# B&R Automation Studio project CentralEne
Automation Studio 4.4.4.112; technology packages: Acp10Arnc0 3.18.2, mapp 1.64.1, mappControl 5.1.0, mappView 5.1.1

## Configuration Central

CPU X20CP1301, AutomationRuntime F4.44, Build 4.1.2, Vc V4.44.0

### Task classes (Cpu.sw)
```
Cyclic#6:
  acionaSina <- Programa.acionaSinais.prg
  preparaDet <- Programa.preparaDetectores.prg
Cyclic#7:
  transmiteD <- Programa.transmiteDetectores.prg
DataObjects: Acp10sys
VcDataObjects: Visu <- Programa.Visu.dob
Binaries: TCData, vccalarm, vcnet, vcrt, vcpkat, vcctext, vctcal, vcfile, vcgclass, vcctrend, Visu03, vcpdsw, arial, vccbmp, vcmgr, vcchspot, vcdsloc, vcfntttf, Visu02, vccovl, vcshared, arialbd, vcalarm, vccdt, vccline, vccbtn, vcpdvnc, vcbclass, vcpfx20, vcdsint, vccnum, Visu01, mvLoader, udbdef, ashwac, Role, ashwd, arconfig, sysconf, iomap, User, asfw, Acp10map, acp10cfg, vcpfar00
Libraries: AsHttp, runtime, standard, LoopConR, sys_lib, brsystem, Acp10par, NcGlobal, Acp10man, asieccon, astime, vcresman, fileio, ashw, dataobj, powerlnk
```

### Hardware
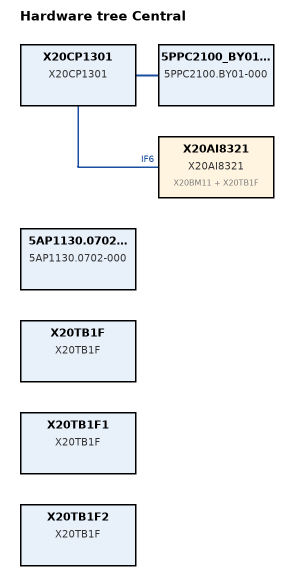
```
5AP1130.0702-000 : 5AP1130.0702-000 v1.3.0.0
  Terminal = true
  Mode = Manual
  InternetAddress = 172.21.12.120
  DefaultGateway = 172.21.12.2
  SubnetMask = 255.255.255.0
5PPC2100_BY01_000 : 5PPC2100.BY01-000 v1.2.9.0  [IF3 -> X20CP1301.IF2 [Cable Type=PowerlinkCable, Length=10, Version=1.0.0.2]; SY -> 5AP1130.0702-000.SY1]
  Connector IF3
  Terminal = true
X20AI8321 : X20AI8321 v1.3.0.0  [SS1 -> X20TB1F3.SS; SL -> X20BM11.SL1]
  LowerLimit = 0
  ChannelType01 = 4 to 20mA
  ChannelType02 = 4 to 20mA
  ChannelType03 = 4 to 20mA
  ChannelType04 = 4 to 20mA
  ChannelType05 = 4 to 20mA
X20BM11 : X20BM11 v1.0.0.1  [X2X1 -> X20CP1301.IF6]
X20CP1301 : X20CP1301 v1.6.1.0  [X1 -> X1.SL; X2 -> X2.SL; X3 -> X3.SL]
  Module X1 (Type=X1, Virtual=true, Version=1.6.1.0)
    Connection (Connector=SS1, TargetModule=X20TB1F, TargetConnector=SS)
    Connection (Connector=SL, TargetModule=X20CP1301, TargetConnector=X1)
  Module X2 (Type=X2, Virtual=true, Version=1.6.1.0)
    Connection (Connector=SS1, TargetModule=X20TB1F1, TargetConnector=SS)
    Connection (Connector=SL, TargetModule=X20CP1301, TargetConnector=X2)
  Module X3 (Type=X3, Virtual=true, Version=1.6.1.0)
    Connection (Connector=SS1, TargetModule=X20TB1F2, TargetConnector=SS)
    Connection (Connector=SL, TargetModule=X20CP1301, TargetConnector=X3)
  Connector IF2:
    ActivateDevice = 1
    HostName = loga
    Mode = Manual
    InternetAddress = 172.21.12.119
    SubnetMask = 255.255.255.0
    Vnc1
    VncVcObjectName1 = Visu
    VncKeyMappingFile1 = VC\PS2-Keyboard.dis
    VncAuthentication1 = 1
    VncPasswordViewOnly1 = v
    VncPasswordViewControl1 = c
  ConfigurationID = CentralEne_Central
  EthernetDefaultGateway = 172.21.12.2
  ActivateDns = 1
  DnsServer1 = 172.21.4.143
X20TB1F : X20TB1F v1.0.0.0
X20TB1F1 : X20TB1F v1.0.0.0
X20TB1F2 : X20TB1F v1.0.0.0
X20TB1F3 : X20TB1F v1.0.0.0
```

### IoMap.iom - X20CP1301/IoMap.iom
```iecst
VAR_CONFIG
	::preparaDet:aiDG[1] AT %IW."X20AI8321".AnalogInput01;
	::preparaDet:aiDG[2] AT %IW."X20AI8321".AnalogInput02;
	::preparaDet:aiDG[3] AT %IW."X20AI8321".AnalogInput03;
	::preparaDet:aiDG[5] AT %IW."X20AI8321".AnalogInput04;
	::preparaDet:aiDG[4] AT %IW."X20AI8321".AnalogInput05;
	::Estrutura.do01SinVd AT %QX."X3".DigitalOutput01;
	::Estrutura.do02SinAm AT %QX."X3".DigitalOutput02;
	::Estrutura.do03SinVm AT %QX."X3".DigitalOutput03;
	::Estrutura.do04SinVd AT %QX."X3".DigitalOutput04;
	::Estrutura.do05SinAm AT %QX."X3".DigitalOutput05;
	::Estrutura.do06SinVm AT %QX."X3".DigitalOutput06;
	::Estrutura.do07Buzer AT %QX."X3".DigitalOutput07;
	::Estrutura.do08Modem AT %QX."X3".DigitalOutput08;
END_VAR
```

### Acp10cfg.ncc - X20CP1301/Motion/Acp10cfg.ncc
```
NcConfiguration (Version=3.18.2, NcSwId=Acp10)
  ACP10CF1_typ:
    cnt_nettrc_rec_drive = 150
    bufsize_trace_upload = 1200
    tc_nc_man_task = Cyclic #1
    glob_pv_as_ncobject = Yes
    ncsys_dl_broadcast = Yes
    ncsys_dl_acp_reset = Yes
    safemc_log_err_to_ax = Yes
    network_init:
      ncsw_init_execute = Yes
      automatic_execute = No
      node_nr_warning = Yes
      net_err_before_ncact = Yes
    nettrc:
      enter_parsecrec = Yes
      enter_ncaction = Yes
      save_ring_startidx = No
    cam_prof_download:
      cam_dat_dl_parallel = No
      tc_cam_dl_parallel = Task class for NC Manager task
```

## Logical view

Binary libraries used (declarations not repeated): operator, runtime, astime, AsIecCon, AsHttp, standard, LoopConR 4.01.0, sys_lib, brsystem, Acp10par 3.18.2, Acp10man 3.18.2, NcGlobal 3.18.2

### Global.typ - Global data types
```iecst
TYPE
	TipoTransmiter : 	STRUCT
		idTxSoftware : STRING[80];
		txValueDet : REAL;
	END_STRUCT;
	TipoEstruturaDG_type : 	STRUCT
		Estatos : REAL;
		TX : STRING[80];
		visDet : USINT;
		ID : STRING[80] := '1';
		Alarme2 : BOOL;
		Alarme1 : BOOL;
		Area : USINT;
	END_STRUCT;
	TipoEstrutura : 	STRUCT
		DG : {REDUND_UNREPLICABLE} ARRAY[0..MAX_IDX_DETECTORES]OF TipoEstruturaDG_type;
		visDet01 : USINT;
		visDet02 : USINT;
		visDet03 : USINT;
		visDet04 : USINT;
		visDet05 : USINT;
		visSinVd : BOOL;
		visSinAm : BOOL;
		visSinVm : BOOL;
		do01SinVd : BOOL;
		do02SinAm : BOOL;
		do03SinVm : BOOL;
		do04SinVd : BOOL;
		do05SinAm : BOOL;
		do06SinVm : BOOL;
		do08Modem : BOOL;
		do07Buzer : BOOL;
		visNameDG1 : STRING[80];
		visNameDG2 : STRING[80];
		visNameDG3 : STRING[80];
		visNameDG4 : STRING[80];
		visNameDG5 : STRING[80];
		visModemReset : BOOL;
	END_STRUCT;
END_TYPE
```

### Global.var - Global variables
```iecst
VAR
	Transmissao : TipoTransmiter;
	Estrutura : TipoEstrutura;
END_VAR
(*CONTANTES*)
VAR CONSTANT
	MAX_IDX_DETECTORES : USINT := 5;
END_VAR
```


### Program Logical/Programa/preparaDetectores (IEC)

#### Variables.var
```iecst
VAR
	aiDG : ARRAY[0..MAX_IDX_DETECTORES] OF INT;
	LCRScal_DG : ARRAY[0..MAX_IDX_DETECTORES] OF LCRScal;
	uIdx : USINT; (*Contador auxiliar*)
END_VAR
```

#### Main.st
```iecst
PROGRAM _INIT
	(* Prepara o range dos detectores *)

	//Configura detector 1
	Estrutura.DG[1].Area 	:= 2;
	Estrutura.DG[2].Area 	:= 2;
	Estrutura.DG[3].Area 	:= 2;
	Estrutura.DG[4].Area 	:= 1;
	Estrutura.DG[5].Area 	:= 2;

	Estrutura.DG[1].ID		:= '73';
	Estrutura.DG[2].ID		:= '74';
	Estrutura.DG[3].ID		:= '75';
	Estrutura.DG[4].ID		:= '72';
	Estrutura.DG[5].ID		:= '76';

	LCRScal_DG[1].x1 := 0.0;	 //x1 e x2 não pode ser alterado, y1 e y2 é o range do detector
	LCRScal_DG[1].y1 := 0.0;
	LCRScal_DG[1].x2 := 32767.0;
	LCRScal_DG[1].y2 := 50.0;

	LCRScal_DG[2].x1 := 0.0;	 //x1 e x2 não pode ser alterado, y1 e y2 é o range do detector
	LCRScal_DG[2].y1 := 0.0;
	LCRScal_DG[2].x2 := 32767.0;
	LCRScal_DG[2].y2 := 100.0;

	LCRScal_DG[3].x1 := 0.0;	 //x1 e x2 não pode ser alterado, y1 e y2 é o range do detector
	LCRScal_DG[3].y1 := 0.0;
	LCRScal_DG[3].x2 := 32767.0;
	LCRScal_DG[3].y2 := 1000.0;

	LCRScal_DG[4].x1 := 0.0;	 //x1 e x2 não pode ser alterado, y1 e y2 é o range do detector
	LCRScal_DG[4].y1 := 0.0;
	LCRScal_DG[4].x2 := 32767.0;
	LCRScal_DG[4].y2 := 1000.0;

	LCRScal_DG[5].x1 := 0.0;	 //x1 e x2 não pode ser alterado, y1 e y2 é o range do detector
	LCRScal_DG[5].y1 := 0.0;
	LCRScal_DG[5].x2 := 32767.0;
	LCRScal_DG[5].y2 := 100.0;

END_PROGRAM

PROGRAM _CYCLIC

	FOR uIdx := 0 TO MAX_IDX_DETECTORES BY 1 DO

		(* Converte em numero real os valores da entrada analogica *)
		LCRScal_DG[uIdx].x := INT_TO_REAL(aiDG[uIdx]);

		(* Chama o bloco de função e declara nas variaveis os resultados *)
		LCRScal_DG[uIdx]();
		Estrutura.DG[uIdx].Estatos 	:= LCRScal_DG[uIdx].y;
		Estrutura.DG[uIdx].TX		:= REAL_TO_STRING (Estrutura.DG[uIdx].Estatos * 100000);

	END_FOR;

END_PROGRAM
```

### Program Logical/Programa/transmiteDetectores (IEC)

#### Types.typ
```iecst
TYPE
	MaqEstados_enum :
		(
		HTTP_STEP_DESABILITADO := 0,
		HTTP_STEP_CONCATENA,
		HTTP_STEP_ENVIA,
		HTTP_STEP_DELAY,
		HTTP_STEP_PROXIMO_DG,
		HTTP_STEP_CONCLUIDO,
		HTTP_STEP_ABORTA,
		HTTP_STEP_ERRO
		);
END_TYPE
```

#### Variables.var
```iecst
VAR
	Dosend : BOOL := TRUE;
	Doenable : BOOL := TRUE; (*Enables FUB Instance*)
END_VAR
VAR CONSTANT
	Host : STRING[80] := '201.6.243.3';
	HostPort : UINT := 8090;
END_VAR
VAR
	Responsedata : STRING[80];
	uri : STRING[80];
	input : BOOL;
	output : BOOL;
	elapsedTime : TIME;
END_VAR
(*Insert your comment here.*)
VAR
	eStep : MaqEstados_enum;
	iDG : USINT; (*Index atual do DG a ser enviado*)
	sAuxiliar : STRING[80];
	httpClient_0 : httpClient;
	bEnviar : BOOL; (*Comando para iniciar envio*)
	TON_0 : TON;
	Resposta : STRING[80];
END_VAR
```

#### Main.st
```iecst
PROGRAM _INIT

	uri     := '/api/historic/SaveByPositionUid2';

	httpClient_0.pHost 				:= ADR (Host);
	httpClient_0.hostPort			:= HostPort;
	httpClient_0.method 			:= httpMETHOD_GET;
	httpClient_0.option 			:= httpOPTION_HTTP_11;
	httpClient_0.pResponseData 		:= ADR (Responsedata);
	httpClient_0.responseDataSize	:= SIZEOF (Responsedata);
	httpClient_0.pUri    			:= ADR (sAuxiliar);

	TON_0.PT := T#15s;

END_PROGRAM

PROGRAM _CYCLIC

	CASE eStep OF

		HTTP_STEP_DESABILITADO:

			bEnviar := TRUE;

			IF(bEnviar)THEN

				//Reseta comando
				bEnviar := FALSE;
				iDG := 1;

				eStep := HTTP_STEP_CONCATENA;

			END_IF

		HTTP_STEP_CONCATENA:

			sAuxiliar				:= CONCAT(uri, CONCAT('/', CONCAT(Estrutura.DG[iDG].ID, CONCAT('/', Estrutura.DG[iDG].TX))));
			httpClient_0.enable		:= TRUE;
			httpClient_0.send		:= TRUE;

			eStep := HTTP_STEP_ENVIA;

		HTTP_STEP_ENVIA:

			//Checa status do bloco
			IF(httpClient_0.status <> 65535)THEN

				IF(httpClient_0.status = 0)THEN

					//Reseta comandos
					httpClient_0.send	:= FALSE;
					TON_0.IN := TRUE;

					eStep := HTTP_STEP_DELAY;
				ELSE
					eStep := HTTP_STEP_ERRO;
				END_IF
			ELSE
				eStep := HTTP_STEP_ERRO;
			END_IF

		HTTP_STEP_DELAY:

			IF(TON_0.Q)THEN

				TON_0.IN := FALSE;
				eStep := HTTP_STEP_PROXIMO_DG;

			END_IF

		HTTP_STEP_PROXIMO_DG:

			iDG := iDG + 1;

			IF(iDG > MAX_IDX_DETECTORES)THEN
				eStep := HTTP_STEP_CONCLUIDO;
			ELSE
				eStep := HTTP_STEP_CONCATENA;
			END_IF

		HTTP_STEP_CONCLUIDO:

			httpClient_0.enable := FALSE;
			httpClient_0.send	:= FALSE;
			TON_0.IN := FALSE;

			eStep := HTTP_STEP_DESABILITADO;

		HTTP_STEP_ABORTA:

			//Reseta blocos
			httpClient_0.enable := FALSE;
			httpClient_0.send	:= FALSE;
			TON_0.IN := FALSE;
			eStep := HTTP_STEP_DESABILITADO;

		HTTP_STEP_ERRO:

			//Reseta blocos
			httpClient_0.enable := FALSE;
			httpClient_0.send	:= FALSE;
			TON_0.IN := FALSE;
			eStep := HTTP_STEP_DESABILITADO;

	END_CASE;

	//Chamada de execução do bloco de função
	httpClient_0();
	TON_0();

END_PROGRAM

PROGRAM _EXIT
	(* Release Client instance *)
	httpClient_0(enable := 0, send := 0);
END_PROGRAM
```

### Program Logical/Programa/acionaSinais (IEC)

#### Main.st
```iecst
PROGRAM _INIT
	(*Prepara os sinalizador e IHM para luz verde acionada*)

	Estrutura.do01SinVd := 1; // Aciona a luz verde do sinalizador
	Estrutura.do02SinAm := 0; // Apaga a luz amarela da sinaleira
	Estrutura.do03SinVm := 0; // Apaga a luz Vermelha da sinaleira
	Estrutura.do04SinVd := 1; // Aciona a luz verde do sinalizador
	Estrutura.do05SinAm := 0; // Apaga a luz amarela da sinaleira
	Estrutura.do06SinVm := 0; // Apaga a luz Vermelha da sinaleira
	Estrutura.do07Buzer := 0;
	Estrutura.visSinVd := 1; //Aciona a luz verde da IHM
END_PROGRAM

PROGRAM _CYCLIC

	(************************************************************
	Checa os limetes de alarmes inferior e superior DO detector 01
	e faz os acionamentos dos sinalizadores de acordo com os
	limites.
	*************************************************************)

	IF Estrutura.DG[1].Estatos < 8 THEN
		Estrutura.visDet01 := 0;
		Estrutura.visSinVd := 1;
		Estrutura.DG[1].Alarme1	:= 0;
		Estrutura.DG[1].Alarme2	:= 0;

	ELSIF Estrutura.DG[1].Estatos >= 8  AND Estrutura.DG[1].Estatos < 12  THEN
		Estrutura.visDet01 := 1;
		Estrutura.DG[1].Alarme1	:= 1;

	ELSIF Estrutura.DG[1].Estatos >= 12  THEN
		Estrutura.visDet01 := 2;
		Estrutura.DG[1].Alarme1	:= 0;
		Estrutura.DG[1].Alarme2	:= 1;

	END_IF

	(************************************************************
	Checa os limetes de alarmes inferior e superior DO detector 02
	e faz os acionamentos dos sinalizadores de acordo com os
	limites.
	*************************************************************)

	IF Estrutura.DG[2].Estatos < 39 THEN
		Estrutura.visDet02 := 0;
		Estrutura.DG[2].Alarme1	:= 0;
		Estrutura.DG[2].Alarme2	:= 0;

	ELSIF Estrutura.DG[2].Estatos >= 39  AND Estrutura.DG[2].Estatos < 43  THEN
		Estrutura.visDet02 := 1;
		Estrutura.DG[2].Alarme1	:= 1;

	ELSIF Estrutura.DG[2].Estatos >= 43  THEN
		Estrutura.visDet02 := 2;
		Estrutura.DG[2].Alarme1	:= 0;
		Estrutura.DG[2].Alarme2	:= 1;

	END_IF

	(************************************************************
	Checa os limetes de alarmes inferior e superior DO detector 03
	e faz os acionamentos dos sinalizadores de acordo com os
	limites.
	*************************************************************)

	IF Estrutura.DG[3].Estatos < 20 THEN
		Estrutura.visDet03 := 0;
		Estrutura.DG[3].Alarme1	:= 0;
		Estrutura.DG[3].Alarme2	:= 0;

	ELSIF Estrutura.DG[3].Estatos >= 20  AND Estrutura.DG[3].Estatos < 40  THEN
		Estrutura.visDet03 := 1;
		Estrutura.DG[3].Alarme1	:= 1;

	ELSIF Estrutura.DG[3].Estatos >= 40  THEN
		Estrutura.visDet03 := 2;
		Estrutura.DG[3].Alarme1	:= 0;
		Estrutura.DG[3].Alarme2	:= 1;

	END_IF

	(************************************************************
	Checa os limetes de alarmes inferior e superior DO detector 04
	e faz os acionamentos dos sinalizadores de acordo com os
	limites.
	*************************************************************)

	IF Estrutura.DG[4].Estatos < 39 THEN
		Estrutura.visDet04 := 0;
		Estrutura.DG[4].Alarme1	:= 0;
		Estrutura.DG[4].Alarme2	:= 0;

	ELSIF Estrutura.DG[4].Estatos >= 39  AND Estrutura.DG[4].Estatos < 43  THEN
		Estrutura.visDet04 := 1;
		Estrutura.DG[4].Alarme1	:= 1;

	ELSIF Estrutura.DG[4].Estatos >= 43  THEN
		Estrutura.visDet04 := 2;
		Estrutura.DG[4].Alarme1	:= 0;
		Estrutura.DG[4].Alarme2	:= 1;

	END_IF

	(************************************************************
	Checa os limetes de alarmes inferior e superior DO detector 05
	e faz os acionamentos dos sinalizadores de acordo com os
	limites.
	*************************************************************)

	IF Estrutura.DG[5].Estatos < 10 THEN
		Estrutura.visDet05 := 0;
		Estrutura.DG[5].Alarme1	:= 0;
		Estrutura.DG[5].Alarme2	:= 0;

	ELSIF Estrutura.DG[5].Estatos >= 10  AND Estrutura.DG[5].Estatos < 20  THEN
		Estrutura.visDet05 := 1;
		Estrutura.DG[5].Alarme1	:= 1;

	ELSIF Estrutura.DG[5].Estatos >= 20  THEN
		Estrutura.visDet05 := 2;
		Estrutura.DG[5].Alarme1	:= 0;
		Estrutura.DG[5].Alarme2	:= 1;

	END_IF

	IF Estrutura.DG[1].Alarme1 OR Estrutura.DG[2].Alarme1 OR Estrutura.DG[3].Alarme1 OR Estrutura.DG[5].Alarme1 = 1 THEN
		Estrutura.do01SinVd	:= 0;
		Estrutura.do02SinAm := 1;
		Estrutura.do03SinVm := 0;
		Estrutura.do07Buzer	:= 0;
		Estrutura.visSinAm 	:= 1;
		Estrutura.visSinVd	:= 0;
		Estrutura.visSinVm	:= 0;

	ELSIF Estrutura.DG[4].Alarme1 = 1 THEN
		Estrutura.do04SinVd	:= 0;
		Estrutura.do05SinAm	:= 1;
		Estrutura.do06SinVm	:= 0;
		Estrutura.do07Buzer	:= 0;
		Estrutura.visSinAm 	:= 1;
		Estrutura.visSinVd	:= 0;
		Estrutura.visSinVm	:= 0;

	ELSIF Estrutura.DG[1].Alarme2 OR Estrutura.DG[2].Alarme2 OR Estrutura.DG[3].Alarme2 OR Estrutura.DG[5].Alarme2 = 1 THEN
		Estrutura.do01SinVd	:= 0;
		Estrutura.do02SinAm	:= 0;
		Estrutura.do03SinVm	:= 1;
		Estrutura.do07Buzer	:= 1;
		Estrutura.visSinVm 	:= 1;
		Estrutura.visSinAm	:= 0;
		Estrutura.visSinVd	:= 0;

	ELSIF Estrutura.DG[4].Alarme2 = 1 THEN
		Estrutura.do04SinVd	:= 0;
		Estrutura.do05SinAm	:= 0;
		Estrutura.do06SinVm	:= 1;
		Estrutura.do07Buzer	:= 1;
		Estrutura.visSinVm 	:= 1;
		Estrutura.visSinAm	:= 0;
		Estrutura.visSinVd	:= 0;

	ELSIF Estrutura.DG[1].Alarme1 OR Estrutura.DG[2].Alarme1 OR Estrutura.DG[3].Alarme1 OR Estrutura.DG[4].Alarme1 OR Estrutura.DG[5].Alarme1 OR Estrutura.DG[1].Alarme2 OR Estrutura.DG[2].Alarme2 OR Estrutura.DG[3].Alarme2 OR Estrutura.DG[4].Alarme2 OR Estrutura.DG[5].Alarme2 = 1 THEN
		Estrutura.do07Buzer := 1;

	ELSE
		Estrutura.visSinVd	:= 1;
		Estrutura.visSinAm	:= 0;
		Estrutura.visSinVm	:= 0;
		Estrutura.do01SinVd	:= 1;
		Estrutura.do02SinAm	:= 0;
		Estrutura.do03SinVm	:= 0;
		Estrutura.do04SinVd	:= 1;
		Estrutura.do05SinAm	:= 0;
		Estrutura.do06SinVm	:= 0;
		Estrutura.do07Buzer	:= 0;

	END_IF

END_PROGRAM

PROGRAM _EXIT
	(* Insert code here *)

END_PROGRAM
```

- Visualisation Logical/Programa/Visu (not shown)
